Staubli VAL3: ComPlc.pgx

program ComPlc()
begin
  do
    // Word de vida de la comunicació entre el robot i el PLC
    if nWordComRobot>10000
      nWordComRobot=0
    endIf
    nWordComRobot=nWordComRobot+1
    aioSet(aoWordComRobot,nWordComRobot)

  until false
end
